Universal Robots PolyScope program: Albert_Samuel_P1.urp

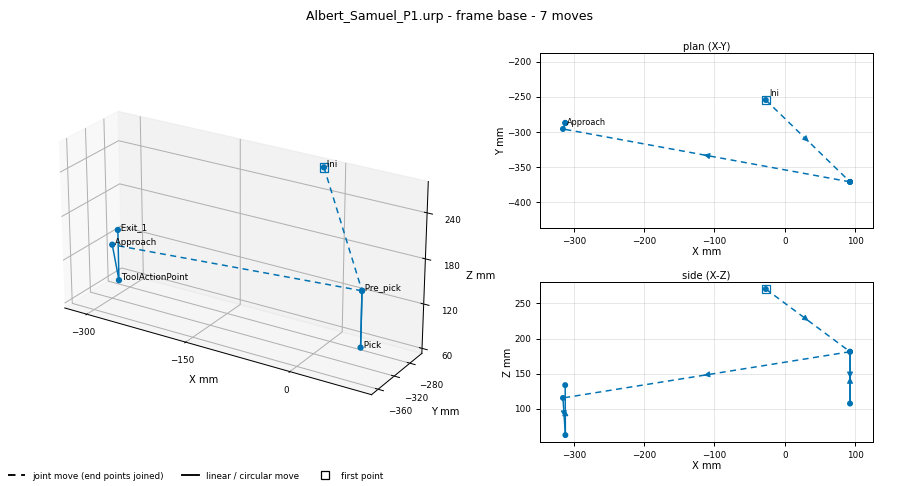
[picture p0: tool path of Albert_Samuel_P1.urp in frame base, 7 of 7 moves have a stored position in this frame; points joined in program order, loops and branches not executed]
Program Albert_Samuel_P1 (installation=default directory=/programs createdIn=5.13.0 lastSavedIn=5.13.0 robotSerialNumber=20195300809)
Calibrated DH parameters: a=[-0.000085, -0.20076, -0.212369, 0.000121, -0.000118, 0]; d=[0.15185, -26.306375, 24.753047, 1.684739, 0.085386, 0.092088]; alpha=[1.572149, -0.00522, -0.011864, 1.571339, -1.571085, 0]; deltaTheta=[0, 0.599885, -0.513355, -0.086555, 0.000006, 0]
InitVariablesNode variables(variable(name=Pallet_1_cnt, expression=1), variable(name=Pallet_1_lct, expression=1), variable(name=Pallet_1_lno, expression=1), variable(name=Pallet_1_sep, expression=False), variable(name=Pallet_1_tct, expression=1), variable(name=var_1, expression=0))
Robot Program (runOnlyOnce=false)
  If var_1<6
    MoveJ speed 60 deg/s, acceleration 80 deg/s^2 (useActiveTCP=true) feature=Base
      Waypoint Ini: TCP in base x=-27.003 y=-254.346 z=270.516 mm, rx=1.4681 ry=2.7067 rz=0.047 rad; joints [-69.643, -80.284, -65.825, -122.305, 93.237, 78.019] deg; TCP offset x=0 y=0 z=150 mm, rx=0 ry=0 rz=0 rad
      Wait DigitalInput pin=digital_in[0]; digitalValue=0
    MoveJ speed 60 deg/s, acceleration 80 deg/s^2 (useActiveTCP=true) feature=Base
      Waypoint Pre_pick: TCP in base x=92.786 y=-370.742 z=181.382 mm, rx=1.2093 ry=2.8313 rz=0.06 rad; joints [-58.756, -104.699, -65.967, -97.685, 93.243, 78.017] deg
    MoveL speed 250 mm/s, acceleration 1200 mm/s^2 (useActiveTCP=true) feature=Base
      Waypoint Pick: TCP in base x=92.769 y=-370.75 z=107.677 mm, rx=1.2093 ry=2.8314 rz=0.06 rad; joints [-58.697, -104.977, -85.499, -77.888, 93.227, 77.844] deg
      URCap Gripper (Robotiq_Grippers, Robotiq Inc.) dataModel(position=100.0, force=0.0, speed=100.0, positionInDouble=100.0, forceInDouble=0.0, speedInDouble=100.0, slaveIds=[9], blocking=true)
      Wait Sleep waitTime=0.5
    MoveL speed 250 mm/s, acceleration 1200 mm/s^2 (useActiveTCP=true) feature=Base
      Waypoint Pre_pick: TCP in base x=92.786 y=-370.742 z=181.382 mm, rx=1.2093 ry=2.8313 rz=0.06 rad; joints [-58.756, -104.699, -65.967, -97.685, 93.243, 78.017] deg
    URCap Palletizing (polyscope-pallet-impl, Universal Robots) dataModel(palletFeature=Base, isPalletizing=true, Length(key=objectHeight value=0.04 unit=M), Variable(key=referencePoint, variable(featureName=referencePoint)), Variable(key=separatorPoint, variable(featureName=separatorPoint)), Variable(key=name, variable(name=Pallet_1)), Variable(key=globalCountingVariable, variable(name=Pallet_1_cnt, initializeExpression=1)), Variable(key=layerCountingVariable, variable(name=Pallet_1_lct, initializeExpression=1)), Variable(key=layerNumberVariable, variable(name=Pallet_1_lno, initializeExpression=1)), Variable(key=handleSeparatorVariable, variable(name=Pallet_1_sep, initializeExpression=False)), Variable(key=totalCountVariable, variable(name=Pallet_1_tct, initializeExpression=1))); state(isChildrenLocked=true)
      URCap Patterns (polyscope-pallet-impl, Universal Robots) state(isChildrenLocked=true)
        URCap Pattern (polyscope-pallet-impl, Universal Robots) dataModel(UUID=6e4f9ea7-2a0c-4e2a-8660-88bd6353c8ad, patternType=GRID, rows=3, columns=2, Variable(key=nameVariable, variable(name=Grid_Pattern_1))); state(isChildrenLocked=true)
          URCap Item (polyscope-pallet-impl, Universal Robots) dataModel(UUID=0ca3edb1-98c4-4fb5-9f13-1936e80c4f11, patternType=GRID, index=0, calibrationDeltaTheta=[2.0871938292282843E-8, 0.5998849625986696, -0.513354759222901, -0.08655474087847535, 6.239817607139875E-6, -6.658617090343766E-8], calibrationA=[-8.52060452638757E-5, -0.2007601879611388, -0.2123691625519033, 1.2105607098011576E-4, -1.1833705743435544E-4, 0.0], calibrationD=[0.15184970286177432, -26.306374840159272, 24.75304670983349, 1.6847390881089916, 0.085385969004481, 0.09208826337351553], calibrationAlpha=[1.5721487795181908, -0.005219907129425837, -0.011864150755780208, 1.5713392161993658, -1.5710853432049288, 0.0], calibrationJointChecksum=[-1860213401, -1859864814, -1494669377, -1328152407, -1329437658, -1329056899], calibrationStatus=2, calibrationValidChecksum=true, baseToFeature=[0.0, 0.0, 0.0, 0.0, 0.0, 0.0], TCPOffset=[8.306240768529705E-7, 2.886863014861518E-6, 0.15001092790240822, -1.1753794529638707E-5, 2.6132015351965907E-5, 6.243426132559199E-6], JointPositions(key=jointpositions, JointPosition(key=[1], Angle(key=pos value=-2.123696 unit=RAD)), JointPosition(key=[2], Angle(key=pos value=-2.077763 unit=RAD)), JointPosition(key=[3], Angle(key=pos value=-1.341345 unit=RAD)), JointPosition(key=[4], Angle(key=pos value=-1.294366 unit=RAD)), JointPosition(key=[5], Angle(key=pos value=1.620641 unit=RAD)), JointPosition(key=[6], Angle(key=pos value=0.999507 unit=RAD))), Variable(key=variable, variable(name=CornerItem_1)))
          URCap Item (polyscope-pallet-impl, Universal Robots) dataModel(UUID=2a8e3ee4-f80c-42ae-a877-885770f2dead, patternType=GRID, index=1, calibrationDeltaTheta=[2.0871938292282843E-8, 0.5998849625986696, -0.513354759222901, -0.08655474087847535, 6.239817607139875E-6, -6.658617090343766E-8], calibrationA=[-8.52060452638757E-5, -0.2007601879611388, -0.2123691625519033, 1.2105607098011576E-4, -1.1833705743435544E-4, 0.0], calibrationD=[0.15184970286177432, -26.306374840159272, 24.75304670983349, 1.6847390881089916, 0.085385969004481, 0.09208826337351553], calibrationAlpha=[1.5721487795181908, -0.005219907129425837, -0.011864150755780208, 1.5713392161993658, -1.5710853432049288, 0.0], calibrationJointChecksum=[-1860213401, -1859864814, -1494669377, -1328152407, -1329437658, -1329056899], calibrationStatus=2, calibrationValidChecksum=true, baseToFeature=[0.0, 0.0, 0.0, 0.0, 0.0, 0.0], TCPOffset=[-6.874487352842573E-6, -1.1820185086219848E-5, 0.1499758581378283, 5.528245288965249E-5, -5.424413080274307E-5, -2.344572786984427E-5], JointPositions(key=jointpositions, JointPosition(key=[1], Angle(key=pos value=-2.477928 unit=RAD)), JointPosition(key=[2], Angle(key=pos value=-1.695243 unit=RAD)), JointPosition(key=[3], Angle(key=pos value=-1.859395 unit=RAD)), JointPosition(key=[4], Angle(key=pos value=-1.180509 unit=RAD)), JointPosition(key=[5], Angle(key=pos value=1.618536 unit=RAD)), JointPosition(key=[6], Angle(key=pos value=0.642757 unit=RAD))), Variable(key=variable, variable(name=CornerItem_2)))
          URCap Item (polyscope-pallet-impl, Universal Robots) dataModel(UUID=1d5d0f69-0b45-4620-8f41-7d718538550d, patternType=GRID, index=2, calibrationDeltaTheta=[2.0871938292282843E-8, 0.5998849625986696, -0.513354759222901, -0.08655474087847535, 6.239817607139875E-6, -6.658617090343766E-8], calibrationA=[-8.52060452638757E-5, -0.2007601879611388, -0.2123691625519033, 1.2105607098011576E-4, -1.1833705743435544E-4, 0.0], calibrationD=[0.15184970286177432, -26.306374840159272, 24.75304670983349, 1.6847390881089916, 0.085385969004481, 0.09208826337351553], calibrationAlpha=[1.5721487795181908, -0.005219907129425837, -0.011864150755780208, 1.5713392161993658, -1.5710853432049288, 0.0], calibrationJointChecksum=[-1860213401, -1859864814, -1494669377, -1328152407, -1329437658, -1329056899], calibrationStatus=2, calibrationValidChecksum=true, baseToFeature=[0.0, 0.0, 0.0, 0.0, 0.0, 0.0], TCPOffset=[1.8814839797112737E-5, 1.5484800934634224E-5, 0.15000608227058868, -6.151561137257471E-5, 1.3118529874725926E-5, 4.6455250630072063E-5], JointPositions(key=jointpositions, JointPosition(key=[1], Angle(key=pos value=-2.239373 unit=RAD)), JointPosition(key=[2], Angle(key=pos value=-1.293764 unit=RAD)), JointPosition(key=[3], Angle(key=pos value=-2.230479 unit=RAD)), JointPosition(key=[4], Angle(key=pos value=-1.19661 unit=RAD)), JointPosition(key=[5], Angle(key=pos value=1.62386 unit=RAD)), JointPosition(key=[6], Angle(key=pos value=0.880593 unit=RAD))), Variable(key=variable, variable(name=CornerItem_3)))
          URCap Item (polyscope-pallet-impl, Universal Robots) dataModel(UUID=0d02e1dd-659f-4aa9-ac90-a67bf41b1536, patternType=GRID, index=3, calibrationDeltaTheta=[2.0871938292282843E-8, 0.5998849625986696, -0.513354759222901, -0.08655474087847535, 6.239817607139875E-6, -6.658617090343766E-8], calibrationA=[-8.52060452638757E-5, -0.2007601879611388, -0.2123691625519033, 1.2105607098011576E-4, -1.1833705743435544E-4, 0.0], calibrationD=[0.15184970286177432, -26.306374840159272, 24.75304670983349, 1.6847390881089916, 0.085385969004481, 0.09208826337351553], calibrationAlpha=[1.5721487795181908, -0.005219907129425837, -0.011864150755780208, 1.5713392161993658, -1.5710853432049288, 0.0], calibrationJointChecksum=[-1860213401, -1859864814, -1494669377, -1328152407, -1329437658, -1329056899], calibrationStatus=2, calibrationValidChecksum=true, baseToFeature=[0.0, 0.0, 0.0, 0.0, 0.0, 0.0], TCPOffset=[-1.8915284640430574E-5, -1.4118147590752583E-5, 0.14998856711004868, 4.374833136581474E-5, -8.918433500904685E-5, -4.414021827290714E-6], JointPositions(key=jointpositions, JointPosition(key=[1], Angle(key=pos value=-1.907683 unit=RAD)), JointPosition(key=[2], Angle(key=pos value=-1.831349 unit=RAD)), JointPosition(key=[3], Angle(key=pos value=-1.705762 unit=RAD)), JointPosition(key=[4], Angle(key=pos value=-1.163046 unit=RAD)), JointPosition(key=[5], Angle(key=pos value=1.621117 unit=RAD)), JointPosition(key=[6], Angle(key=pos value=1.21415 unit=RAD))), Variable(key=variable, variable(name=CornerItem_4)))
      URCap Layers (polyscope-pallet-impl, Universal Robots) dataModel(separators=[false], selectedPatterns=[6e4f9ea7-2a0c-4e2a-8660-88bd6353c8ad])
      URCap At Each Item (polyscope-pallet-impl, Universal Robots) dataModel(selectedPattern=6e4f9ea7-2a0c-4e2a-8660-88bd6353c8ad, selectedPosition=0ca3edb1-98c4-4fb5-9f13-1936e80c4f11, Approach_calibrationDeltaTheta=[2.0871938292282843E-8, 0.5998849625986696, -0.513354759222901, -0.08655474087847535, 6.239817607139875E-6, -6.658617090343766E-8], Approach_calibrationA=[-8.52060452638757E-5, -0.2007601879611388, -0.2123691625519033, 1.2105607098011576E-4, -1.1833705743435544E-4, 0.0], Approach_calibrationD=[0.15184970286177432, -26.306374840159272, 24.75304670983349, 1.6847390881089916, 0.085385969004481, 0.09208826337351553], Approach_calibrationAlpha=[1.5721487795181908, -0.005219907129425837, -0.011864150755780208, 1.5713392161993658, -1.5710853432049288, 0.0], Approach_calibrationJointChecksum=[-1860213401, -1859864814, -1494669377, -1328152407, -1329437658, -1329056899], Approach_calibrationStatus=2, Approach_calibrationValidChecksum=true, Approach_baseToFeature=[0.0, 0.0, 0.0, 0.0, 0.0, 0.0], Approach_TCPOffset=[-1.3081887072941E-5, 6.505236326115327E-6, 0.1500143158434177, -1.1538497718620484E-5, 2.0074936622545474E-5, -1.2255714112036006E-5], Exit_calibrationDeltaTheta=[2.0871938292282843E-8, 0.5998849625986696, -0.513354759222901, -0.08655474087847535, 6.239817607139875E-6, -6.658617090343766E-8], Exit_calibrationA=[-8.52060452638757E-5, -0.2007601879611388, -0.2123691625519033, 1.2105607098011576E-4, -1.1833705743435544E-4, 0.0], Exit_calibrationD=[0.15184970286177432, -26.306374840159272, 24.75304670983349, 1.6847390881089916, 0.085385969004481, 0.09208826337351553], Exit_calibrationAlpha=[1.5721487795181908, -0.005219907129425837, -0.011864150755780208, 1.5713392161993658, -1.5710853432049288, 0.0], Exit_calibrationJointChecksum=[-1860213401, -1859864814, -1494669377, -1328152407, -1329437658, -1329056899], Exit_calibrationStatus=2, Exit_calibrationValidChecksum=true, Exit_baseToFeature=[0.0, 0.0, 0.0, 0.0, 0.0, 0.0], Exit_TCPOffset=[2.197416944543784E-5, -2.185957678624284E-5, 0.1499913546865311, 5.4962914067544664E-5, -2.5631753260448325E-6, 6.515092561217905E-5], currentWizardState=MANUAL, Pose(key=refBaseToFeature, Position(key=posePosition, Length(key=X value=0 unit=M), Length(key=Y value=0 unit=M), Length(key=Z value=0 unit=M)), Rotation(key=poseRotation, Angle(key=RX value=0 unit=RAD), Angle(key=RY value=0 unit=RAD), Angle(key=RZ value=0 unit=RAD))), Pose(key=refPose, Position(key=posePosition, Length(key=X value=-0.311996 unit=M), Length(key=Y value=-0.287365 unit=M), Length(key=Z value=0.06284 unit=M)), Rotation(key=poseRotation, Angle(key=RX value=2.154675 unit=RAD), Angle(key=RY value=2.202301 unit=RAD), Angle(key=RZ value=0.023593 unit=RAD))), JointPositions(key=Approach_jointpositions, JointPosition(key=[1], Angle(key=pos value=-2.095913 unit=RAD)), JointPosition(key=[2], Angle(key=pos value=-2.024348 unit=RAD)), JointPosition(key=[3], Angle(key=pos value=-1.185205 unit=RAD)), JointPosition(key=[4], Angle(key=pos value=-1.466724 unit=RAD)), JointPosition(key=[5], Angle(key=pos value=1.577822 unit=RAD)), JointPosition(key=[6], Angle(key=pos value=0.971373 unit=RAD))), JointPositions(key=Exit_jointpositions, JointPosition(key=[1], Angle(key=pos value=-2.119439 unit=RAD)), JointPosition(key=[2], Angle(key=pos value=-2.01703 unit=RAD)), JointPosition(key=[3], Angle(key=pos value=-1.102831 unit=RAD)), JointPosition(key=[4], Angle(key=pos value=-1.578205 unit=RAD)), JointPosition(key=[5], Angle(key=pos value=1.610331 unit=RAD)), JointPosition(key=[6], Angle(key=pos value=0.974946 unit=RAD))))
        URCap Generated Movements (polyscope-pallet-impl, Universal Robots) state(isChildrenLocked=true)
          MoveJ speed 60 deg/s, acceleration 80 deg/s^2 (useActiveTCP=true) feature=referencePoint
            Waypoint Approach: TCP in base x=-315.416 y=-295.537 z=115.673 mm, rx=2.1121 ry=2.2886 rz=-0.0475 rad; joints [-120.087, -115.987, -67.907, -84.037, 90.403, 55.656] deg; TCP offset x=-0.013 y=0.007 z=150.014 mm, rx=0 ry=0 rz=0 rad; feature pose in base x=-311.996 y=-287.365 z=62.84 mm, rx=2.1547 ry=2.2023 rz=0.0236 rad
          MoveL speed 250 mm/s, acceleration 1200 mm/s^2 (useActiveTCP=true) feature(featureName=referencePoint)
            Waypoint ToolActionPoint: TCP in base x=-311.996 y=-287.365 z=62.84 mm, rx=2.1547 ry=2.2023 rz=0.0236 rad; joints [-121.679, -119.047, -76.853, -74.162, 92.856, 57.268] deg; TCP offset x=0.001 y=0.003 z=150.011 mm, rx=0 ry=0 rz=0 rad
          Folder Tool action
            URCap Gripper (Robotiq_Grippers, Robotiq Inc.) dataModel(position=0.0, force=0.0, speed=100.0, positionInDouble=0.0, forceInDouble=0.0, speedInDouble=100.0, slaveIds=[9], blocking=true)
            Wait Sleep waitTime=0.5
          MoveL speed 250 mm/s, acceleration 1200 mm/s^2 (useActiveTCP=true) feature(featureName=referencePoint)
            Waypoint Exit_1: TCP in base x=-312.265 y=-286.75 z=133.883 mm, rx=2.1234 ry=2.242 rz=-0.004 rad; joints [-121.435, -115.567, -63.188, -90.424, 92.265, 55.86] deg; TCP offset x=0.022 y=-0.022 z=149.991 mm, rx=0.0001 ry=0 rz=0.0001 rad
            var_1 := var_1+1
            If var_1≟6
              Popup Warning (haltProgram=false message=Replace pallet! inputType=Text)
              var_1 := 0
Thread Thread_1 (runOnlyOnce=false)
  If digital_in[0]≟ False  or var_1≟6
    Set DigitalOutput pin=digital_out[0]; digitalValue=0
  Else 
    Set DigitalOutput pin=digital_out[0]; digitalValue=1
